TYPE ST_KNXnetIP_ConnectionHeader :
STRUCT
	nStructureLength			: BYTE;
	nCommunicationChannel		: BYTE;
	nSequenceCounter			: BYTE;
	nReserved					: BYTE;
END_STRUCT
END_TYPE

(* stored: Version 1.1.0.1
   DUT ST_KNXnetIP_ConnectionHeader: Id {acd13b96-f912-4da6-bbd5-760b56551d52} *)
